(* PLC project SafeLOGIC-1, BrAutomation SafeDESIGNER  4.4.0.0 *)
(* stored: companyURL http://www.br-automation.com, creationDateTime Thu Mar 18 11:48:17 2021 *)

PROGRAM Main

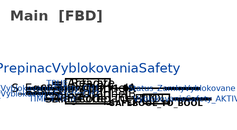
(* FBD diagram, written out as Structured Text *)
PrepinacVyblokovaniaSafety(Activate := TRUE, S_ChannelA := SI_VyblokovanieSafety_CH1, S_ChannelB := SI_VyblokovanieSafety_CH2, DiscrepancyTime := TIME#20ms);
Status_ZamkyVyblokovane := PrepinacVyblokovaniaSafety.S_EquivalentOut;
VyblokovanieSafety_AKTIVNE := SAFEBOOL_TO_BOOL(PrepinacVyblokovaniaSafety.S_EquivalentOut);
END_PROGRAM
